TYPE TupleStruct:
    STRUCT
        field1: REAL;
        field2: REAL;
    END_STRUCT;
END_TYPE
